FUNCTION_BLOCK FB_PressureInputScaling
VAR_INPUT
	nRawInput : INT;
END_VAR
VAR_OUTPUT
	fOutput : LREAL;
END_VAR
VAR
	fRawInput : LREAL;
	fNormalizedInput: LREAL;
	fMinInputValue			: LREAL := 0.0;
	fMaxInputValue			: LREAL := 32767.0;
	fMaxOutputValue 		: LREAL := 400.0;
	fMinOutputValue  		: LREAL := 0.0;			
END_VAR

fRawInput := INT_TO_LREAL(nRawInput);

fNormalizedInput := (fRawInput - fMinInputValue) / (fMaxInputValue - fMinInputValue);

fOutput := LIMIT(fMinOutputValue, fMinOutputValue + fNormalizedInput*(fMaxOutputValue - fMinOutputValue), fMaxOutputValue);

END_FUNCTION_BLOCK

(* stored: Version 1.1.0.1, ProductVersion 3.1.4024.10
   POU FB_PressureInputScaling: Id {b6baeb93-a8de-456f-beee-bdec5c6cc76b}, SpecialFunc None *)
